FUNCTION_BLOCK Exit
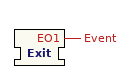
  EVENT_OUTPUT
    EO1;
  END_EVENT
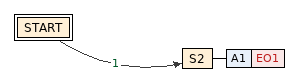
  EC_STATES
    START;
    S2 : A1 -> EO1;
  END_STATES
  EC_TRANSITIONS
    START TO S2 := 1;
  END_TRANSITIONS
  ALGORITHM A1 IN ST:
EXIT;&#38;#10;
  END_ALGORITHM
END_FUNCTION_BLOCK
